// Initialize a ST_ParseContext, building all ST_ParserInternalState from defaults and the given buffer.
FUNCTION F_ParseContextInitializeFromState : ST_ParseContext
VAR_IN_OUT CONSTANT
    stState : ST_ParserInternalState;
END_VAR
VAR_INPUT
    stBuffer : ST_Span;    
END_VAR


F_ParseContextInitializeFromState.stBuffer := stBuffer;
F_ParseContextInitializeFromState.stState  := stState;

END_FUNCTION

(* stored: Version 1.1.0.1
   POU F_ParseContextInitializeFromState: Id {75cd27fb-64c6-4493-9ee6-91cc0b12abeb}, SpecialFunc None *)
